TYPE STATE:
    STRUCT
        curTime: LREAL;
    END_STRUCT;
END_TYPE
